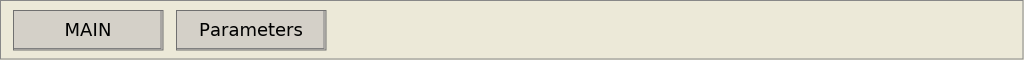
VISUALIZATION Footer  // 1024x60
    Button (13,10 150x40), "MAIN"
        OnMouseClick: change screen: Visualization
    Button (176,10 150x40), "Parameters"
        OnMouseClick: change screen: Footer
END_VISUALIZATION

(* stored: Version 1.1.0.1, ProductVersion 3.1.4024.12
   Visu Footer: Id {4f2f49a3-3e45-4209-9759-e252911f2bf2} *)
